{attribute 'linkalways'} 
{attribute 'no_explicit_call' := 'This FB is a CLASS and must be accessed using methods or properties'}
{attribute 'enable_dynamic_creation'}
FUNCTION_BLOCK _ETcVnSvmSgdClassifierType EXTENDS EnumDatatypeBase
VAR
	localData : ETcVnSvmSgdClassifierType;
	activeData : REFERENCE TO ETcVnSvmSgdClassifierType;
	enumBaseDatatype : _DINT(localData);
END_VAR

METHOD PRIVATE AddLocalEnumeration
VAR_INPUT
	Enumeration : T_MAXSTRING;
	Value : ETcVnSvmSgdClassifierType;
END_VAR
AddEnumeration(Enumeration, Value);
END_METHOD

PROPERTY PUBLIC Address : PVOID
GET
Address := ADR(activeData);
END_GET
END_PROPERTY

METHOD PUBLIC ClearReference
VAR_INPUT
END_VAR
activeData REF= localData;
SetBaseDatatypeReference();
END_METHOD

METHOD PUBLIC Clone : I_Datatype
VAR
    pClone : POINTER TO _ETcVnSvmSgdClassifierType;
END_VAR
pClone := __NEW(_ETcVnSvmSgdClassifierType(InitialValue := Value));
Clone := pClone^;
END_METHOD

METHOD FB_init : BOOL
VAR_INPUT
	bInitRetains : BOOL; // if TRUE, the retain variables are initialized (warm start / cold start)
	bInCopyCode : BOOL;  // if TRUE, the instance afterwards gets moved into the copy code (online change)
	InitialValue : ETcVnSvmSgdClassifierType;
END_VAR
localData := InitialValue;
AddBaseDatatype(enumBaseDatatype);
ClearReference();

AddLocalEnumeration('TCVN_SSCT_SGD', ETcVnSvmSgdClassifierType.TCVN_SSCT_SGD);
AddLocalEnumeration('TCVN_SSCT_ASGD', ETcVnSvmSgdClassifierType.TCVN_SSCT_ASGD);
END_METHOD

PROPERTY PUBLIC Identifier : T_MAXSTRING
GET
Identifier := 'ETcVnSvmSgdClassifierType';
END_GET
END_PROPERTY

METHOD IsEnumeratorValueEqual : BOOL
VAR_INPUT
	Enumerator : I_KeyValueForwardEnumerator;
END_VAR
VAR
	storedValue : ETcVnSvmSgdClassifierType;
END_VAR
IF NOT Enumerator.TryGet(storedValue) THEN
	RETURN;
END_IF

IsEnumeratorValueEqual := storedValue = activeData;
END_METHOD

METHOD PUBLIC MakeReferenceTo
VAR_INPUT
	ReferenceTarget : REFERENCE TO ETcVnSvmSgdClassifierType;
END_VAR
activeData REF= ReferenceTarget;
SetBaseDatatypeReference();
END_METHOD

METHOD PROTECTED SetBaseDatatypeReference
VAR_INPUT
END_VAR
enumBaseDatatype.MakeReferenceTo(activeData);
END_METHOD

PROPERTY PUBLIC Size : UDINT
GET
Size := SIZEOF(activeData);
END_GET
END_PROPERTY

METHOD TryMakeReferenceTo : BOOL
VAR_INPUT
	Target : I_Datatype;
END_VAR
VAR
	targetAsEnum : I_EnumDatatype;
	pTargetData : POINTER TO ETcVnSvmSgdClassifierType;
END_VAR
IF NOT Target.TryResolveAsEnumDatatype(targetAsEnum) THEN
	RETURN;
END_IF

IF targetAsEnum.Identifier <> Identifier THEN
	RETURN;
END_IF

pTargetData := Target.Address;
activeData REF= pTargetData^;
SetBaseDatatypeReference();
TryMakeReferenceTo := TRUE;
END_METHOD

PROPERTY PUBLIC Value : ETcVnSvmSgdClassifierType
GET
Value := activeData;
END_GET
SET
activeData := Value;
END_SET
END_PROPERTY

END_FUNCTION_BLOCK

(* stored: Version 1.1.0.1
   POU _ETcVnSvmSgdClassifierType: Id {7e52b89b-969d-4558-8d99-7bc34ad79b1a}, SpecialFunc None
   Folder Constructor: Id {921e8e1a-f786-434c-ac73-e31e2c91aee0}
   Folder Private: Id {445cec4c-dea5-4c10-9c64-bf2f0f71b84e}
   Folder Protected: Id {cf65b8c0-4ea4-4fc6-838a-9a58837d24de}
   Method AddLocalEnumeration: Id {d0c490a3-8463-4fc6-9dca-49f1acf282c8}
   Property Address: Id {1b8fd09c-2bc9-43ce-b20a-447a55dfe225}
   Get Get: Id {a86b3ac8-9158-4c6e-bf4a-e60aa08b5ec6}
   Method ClearReference: Id {4f905269-7227-4723-8489-06fc153bb599}
   Method Clone: Id {aab2d187-d6dd-4d92-9a3f-8538c0d0077c}
   Method FB_init: Id {3e53fe89-fb2d-49d4-82d7-2d5813b33874}
   Property Identifier: Id {f2489b64-3209-43fc-ae82-7d82ff2aa0b2}
   Get Get: Id {2ae85af5-5572-4c5f-8c8e-33573012eb06}
   Method IsEnumeratorValueEqual: Id {be46814a-d8ab-4df9-9451-94ac22d31661}
   Method MakeReferenceTo: Id {18be9cd8-d10d-435b-abf4-8092e139cae3}
   Method SetBaseDatatypeReference: Id {b42d27ef-0603-4d41-870a-7b2b052488b1}
   Property Size: Id {5494959c-8b5e-4df6-9931-28bdeb588eac}
   Get Get: Id {ca811418-0d73-41f4-aca6-d2af1455525b}
   Method TryMakeReferenceTo: Id {95841b1b-e432-4833-963f-23e048f27a27}
   Property Value: Id {1b015c5f-4795-4c0d-8885-69e9220e01d6}
   Get Get: Id {d435c98e-d326-4fb7-a45f-6ae516a592de}
   Set Set: Id {60e51b01-5f52-4d12-9a95-9c7d11ea271f} *)
